FUNCTION_BLOCK SifbAmmeter
  (* Standard: 61499-2 *)
  (* Version 0.1, 2019-00-29, hpea485, UOA *)
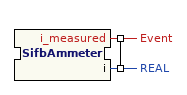
  EVENT_OUTPUT
    i_measured WITH i;
  END_EVENT
  VAR_OUTPUT
    i : REAL;
  END_VAR
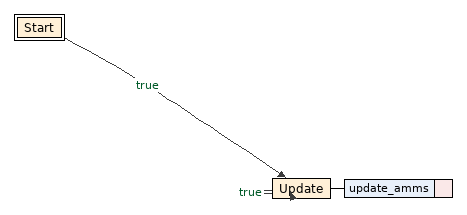
  EC_STATES
    Start;
    Update : update_amms;
  END_STATES
  EC_TRANSITIONS
    Start TO Update := true;
    Update TO Update := true;
  END_TRANSITIONS
  ALGORITHM update_amms IN C:
int sw_ammh = (SWITCHES & 0b1000 != 0);

if(sw_ammh == 1 && int(me->i_set) != 300) {
	//switch is pressed
	me->i = 300.0;
	me->outputEvents.event.i_change = 1;
}
if(sw_ammh == 0 && int(me->i_set) != 5) {
	//switch is pressed
	me->i_set = 5.0;
	me->outputEvents.event.i_change = 1;
}
  END_ALGORITHM
END_FUNCTION_BLOCK
